// Mitsubishi GX Works2 project: PLC_Group12   PLC: FX3G

// global labels: Global1
VAR_GLOBAL
  switch7 AT X007 : BOOL;
  input_chocolate AT D1100 : REAL;
  reg_chocolate_container AT D1110 : REAL;
  reg_nuts_container AT D1112 : REAL;
  input_nuts AT D1102 : REAL;
  reg_pistachio_container AT D1114 : REAL;
  reg_kadaif_container AT D1116 : REAL;
  input_pistachio AT D1104 : REAL;
  input_kadaif AT D1106 : REAL;
  light7 AT Y007 : BOOL;
END_VAR
VAR_GLOBAL CONSTANT
  min_chocolate : REAL := 400.0;
  min_nuts : REAL := 100.0;
  min_pistachio : REAL := 120.0;
  min_kadaif : REAL := 60.0;
END_VAR
VAR_GLOBAL
  check_quantity AT M0 : BOOL;
  switch1 AT X001 : BOOL;
  melting_container AT D1120 : REAL;
  melting_process AT Y001 : BOOL;
  switch2 AT X002 : BOOL;
  switch3 AT X003 : BOOL;
  pouring AT TC1 : BOOL;
END_VAR
VAR_GLOBAL CONSTANT
  pouring_time : INT := 40;
END_VAR
VAR_GLOBAL
  pouring_light AT Y002 : BOOL;
  end_pouring AT TS1 : BOOL;
  switch4 AT X004 : BOOL;
  analog_input_1 AT D8280 : INT;
END_VAR
VAR_GLOBAL CONSTANT
  input_normalize : REAL := 400.0;
END_VAR
VAR_GLOBAL
  chocolate_choice AT D2000 : REAL;
END_VAR
VAR_GLOBAL CONSTANT
  min_choc_nuts : REAL;
  max_choc_nuts : REAL := 5.0;
END_VAR
VAR_GLOBAL
  choc_nuts_light AT M1 : BOOL;
END_VAR
VAR_GLOBAL CONSTANT
  max_choc_dubai : REAL := 10;
  min_choc_dubai : REAL := 5;
END_VAR
VAR_GLOBAL
  choc_dubai_light AT M2 : BOOL;
  pouring_container AT D1122 : REAL;
END_VAR
VAR_GLOBAL CONSTANT
  nuts_filler_for_nuts_choc : REAL := 100.0;
  pistachio_filler_for_nuts_choc : REAL := 100.0;
  nut_filler_for_dubai_choc : REAL := 20.0;
  pistachio_filler_for_dubai_choc : REAL := 120.0;
  kadaif_filler_for_dubai_choc : REAL := 60.0;
END_VAR
VAR_GLOBAL
  blinking3 AT M3 : BOOL;
  light3 AT Y003 : BOOL;
  blinking_switch_3 AT TS3 : BOOL;
  blinking_time_3 AT TC3 : BOOL;
  blinking_time_4 AT TC4 : BOOL;
END_VAR
VAR_GLOBAL CONSTANT
  blinking_time_limit_3 : INT := 10;
  blinking_time_limit_4 : INT := 10;
END_VAR
VAR_GLOBAL
  light4 AT Y004 : BOOL;
  blinking_switch_4 AT TS4 : BOOL;
  blinking_help_light_4 AT M4 : BOOL;
  blinking_help_light_5 AT TS5 : BOOL;
END_VAR
VAR_GLOBAL CONSTANT
  total_blinking_time : INT := 50;
END_VAR
VAR_GLOBAL
  blinking_time_5 AT TC5 : BOOL;
  switch6 AT X006 : BOOL;
  light6 AT Y006 : BOOL;
  cooling_switch AT TS6 : BOOL;
  cool_timer AT TC6 : BOOL;
END_VAR
VAR_GLOBAL CONSTANT
  cool_limit_time : WORD := 30;
END_VAR
VAR_GLOBAL
  switch0 AT X000 : BOOL;
  bars_counter AT CC0 : BOOL;
  bars_counter_switch AT CS0 : BOOL;
END_VAR
VAR_GLOBAL CONSTANT
  bars_limit : WORD := 4;
END_VAR
VAR_GLOBAL
  package_of_four_counter AT D1300 : REAL;
END_VAR
VAR_GLOBAL CONSTANT
  add_one_package : REAL := 1.0;
END_VAR
VAR_GLOBAL
  analog_output AT D8282 : INT;
END_VAR
VAR_GLOBAL CONSTANT
  zero_reset : REAL;
END_VAR
VAR_GLOBAL
  switch5 AT X005 : BOOL;
END_VAR
VAR_GLOBAL CONSTANT
  reset_chocolate_choice : REAL := 15.0;
END_VAR
VAR_GLOBAL
  process_1_done AT M11 : BOOL;
END_VAR
VAR_GLOBAL CONSTANT
  output_normalize : REAL := 40.0;
END_VAR
VAR_GLOBAL
  process_2_done AT M12 : BOOL;
  process_3_done AT M13 : BOOL;
  process_4_done AT M14 : BOOL;
  process_0_done AT M10 : BOOL;
  process_6_done AT M16 : BOOL;
  end_pouring_light AT M21 : BOOL;
  blinking_light_end AT M20 : BOOL;
  cool_light_end AT M22 : BOOL;
  choice_out_of_range AT M40 : BOOL;
  bars_packaging_light AT Y005 : BOOL;
END_VAR
VAR_GLOBAL CONSTANT
  devide_10_output : REAL := 10;
END_VAR

// task Task_01 (event TRUE, interval 0, priority 31): POU_01

PROGRAM POU_01
(* structured ladder/FBD written out as ST: instructions are called as NAME(EN, inputs, outputs); _pN, _eN, _tN stand for wires *)
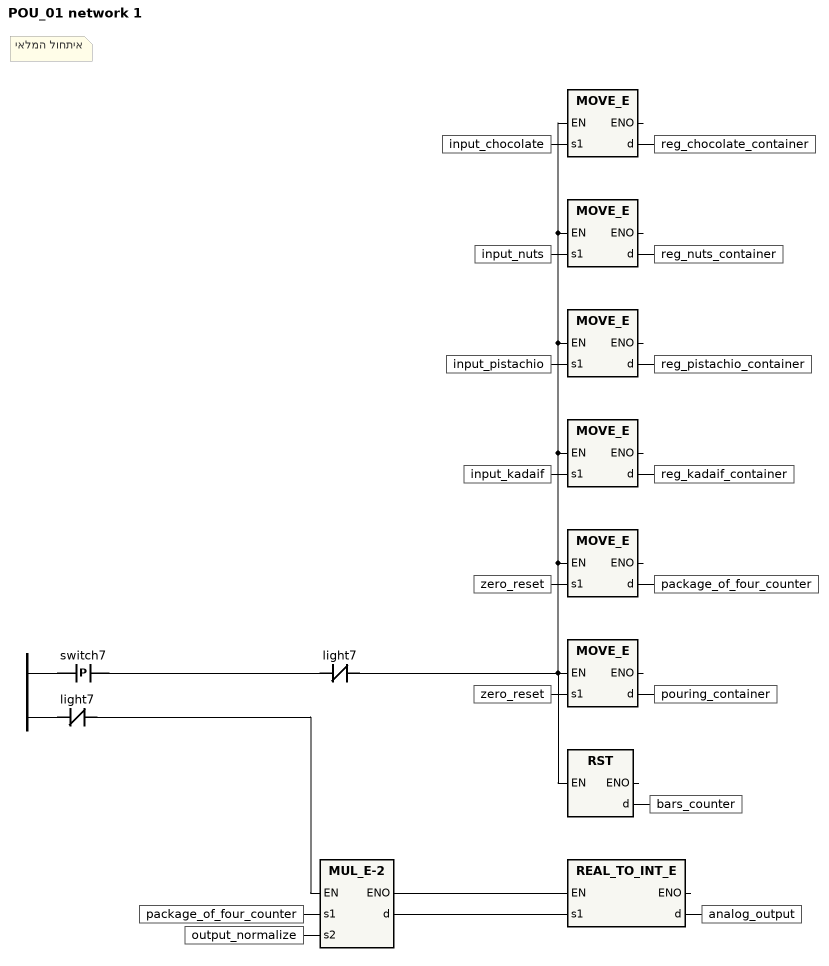
(* network 1 *)
(* איתחול המלאי *)
_p1 := LDP(TRUE, switch7) AND NOT light7;
MOVE_E(_p1, input_chocolate, reg_chocolate_container);
MOVE_E(_p1, input_nuts, reg_nuts_container);
MOVE_E(_p1, input_pistachio, reg_pistachio_container);
MOVE_E(_p1, input_kadaif, reg_kadaif_container);
MOVE_E(_p1, zero_reset, package_of_four_counter);
MOVE_E(_p1, zero_reset, pouring_container);
RST(_p1, bars_counter);
_e3 := MUL_E(NOT light7, package_of_four_counter, output_normalize, _t2);
REAL_TO_INT_E(_e3, _t2, analog_output);
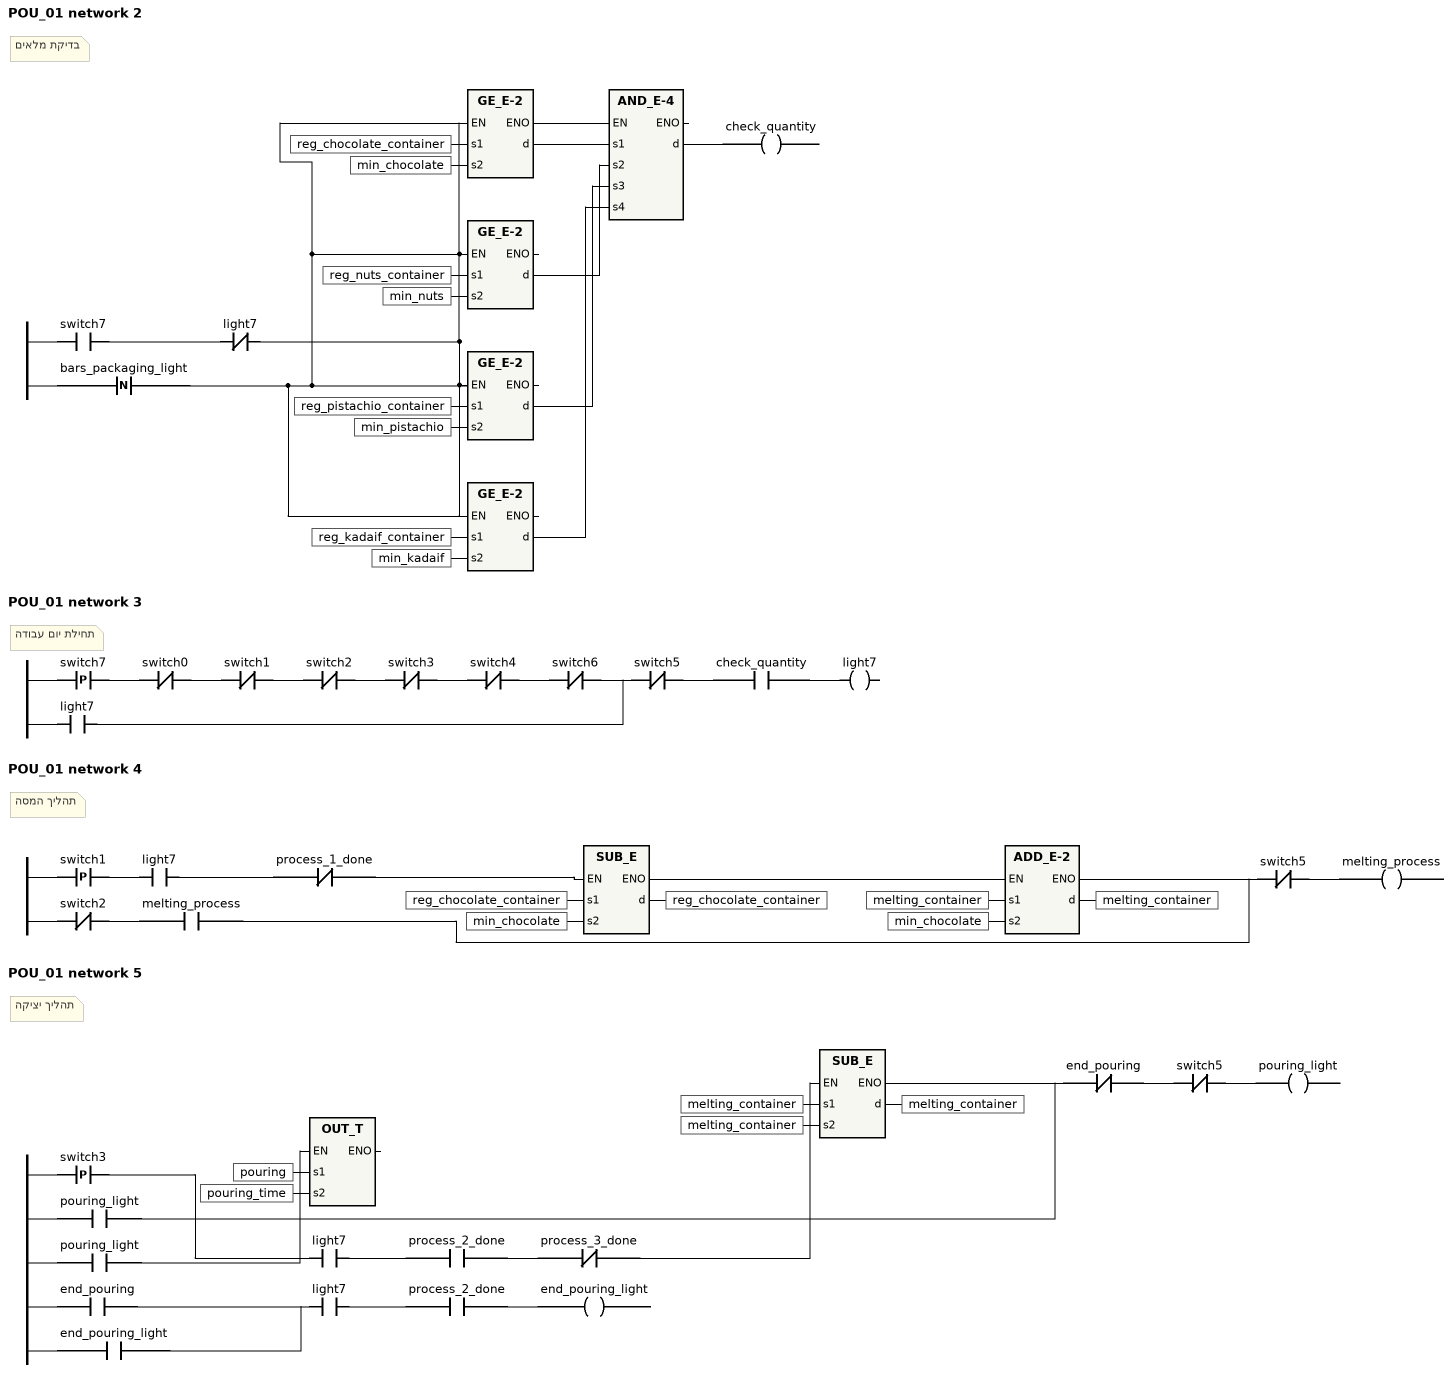
(* network 2 *)
(* בדיקת מלאים *)
_p1 := (switch7 AND NOT light7) OR LDF(TRUE, bars_packaging_light);
_e3 := GE_E(_p1, reg_chocolate_container, min_chocolate, _t2);
GE_E(_p1, reg_nuts_container, min_nuts, _t4);
GE_E(_p1, reg_pistachio_container, min_pistachio, _t5);
GE_E(_p1, reg_kadaif_container, min_kadaif, _t6);
AND_E(_e3, _t2, _t4, _t5, _t6, _t7);
check_quantity := _t7;
(* network 3 *)
(* תחילת יום עבודה *)
light7 := (((LDP(TRUE, switch7) AND NOT switch0 AND NOT switch1 AND NOT switch2 AND NOT switch3 AND NOT switch4 AND NOT switch6) OR light7) AND NOT switch5) AND check_quantity;
(* network 4 *)
(* תהליך המסה *)
_e1 := SUB_E(LDP(TRUE, switch1) AND light7 AND NOT process_1_done, reg_chocolate_container, min_chocolate, reg_chocolate_container);
_e2 := ADD_E(_e1, melting_container, min_chocolate, melting_container);
melting_process := (_e2 OR (NOT switch2 AND melting_process)) AND NOT switch5;
(* network 5 *)
(* תהליך יציקה *)
_e1 := SUB_E(LDP(TRUE, switch3) AND light7 AND process_2_done AND NOT process_3_done, melting_container, melting_container, melting_container);
pouring_light := ((_e1 OR pouring_light) AND NOT end_pouring) AND NOT switch5;
OUT_T(pouring_light, pouring, pouring_time);
end_pouring_light := ((end_pouring OR end_pouring_light) AND light7) AND process_2_done;
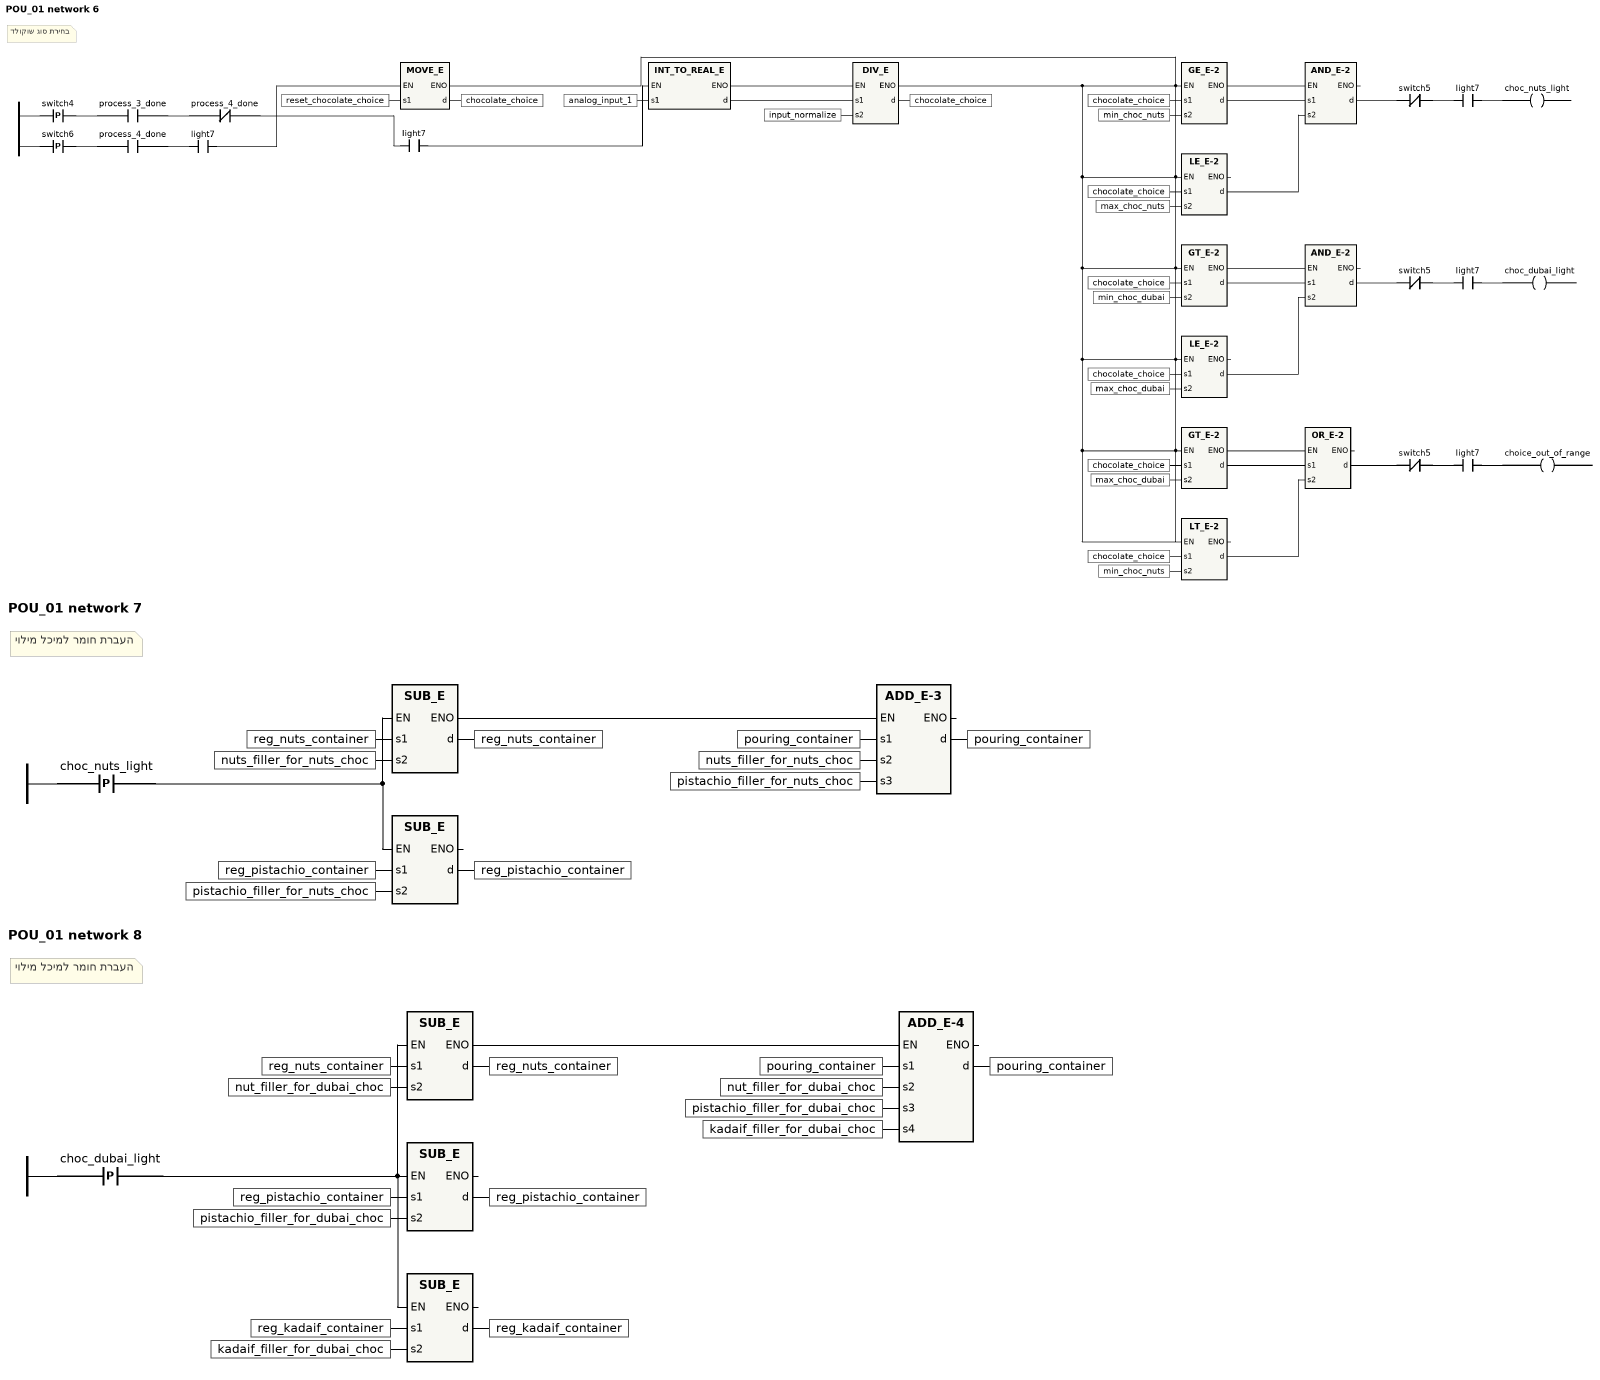
(* network 6 *)
(* בחירת סוג שוקולד *)
_e2 := INT_TO_REAL_E(LDP(TRUE, switch4) AND process_3_done AND NOT process_4_done AND light7, analog_input_1, _t1);
_e3 := DIV_E(_e2, _t1, input_normalize, chocolate_choice);
_e4 := MOVE_E(LDP(TRUE, switch6) AND process_4_done AND light7, reset_chocolate_choice, chocolate_choice);
_p5 := _e3 OR _e4;
_e7 := GE_E(_p5, chocolate_choice, min_choc_nuts, _t6);
LE_E(_p5, chocolate_choice, max_choc_nuts, _t8);
AND_E(_e7, _t6, _t8, _t9);
choc_nuts_light := _t9 AND NOT switch5 AND light7;
_e11 := GT_E(_p5, chocolate_choice, min_choc_dubai, _t10);
LE_E(_p5, chocolate_choice, max_choc_dubai, _t12);
AND_E(_e11, _t10, _t12, _t13);
choc_dubai_light := _t13 AND NOT switch5 AND light7;
_e15 := GT_E(_p5, chocolate_choice, max_choc_dubai, _t14);
LT_E(_p5, chocolate_choice, min_choc_nuts, _t16);
OR_E(_e15, _t14, _t16, _t17);
choice_out_of_range := _t17 AND NOT switch5 AND light7;
(* network 7 *)
(* העברת חומר למיכל מילוי *)
_p1 := LDP(TRUE, choc_nuts_light);
_e2 := SUB_E(_p1, reg_nuts_container, nuts_filler_for_nuts_choc, reg_nuts_container);
ADD_E(_e2, pouring_container, nuts_filler_for_nuts_choc, pistachio_filler_for_nuts_choc, pouring_container);
SUB_E(_p1, reg_pistachio_container, pistachio_filler_for_nuts_choc, reg_pistachio_container);
(* network 8 *)
(* העברת חומר למיכל מילוי *)
_p1 := LDP(TRUE, choc_dubai_light);
_e2 := SUB_E(_p1, reg_nuts_container, nut_filler_for_dubai_choc, reg_nuts_container);
ADD_E(_e2, pouring_container, nut_filler_for_dubai_choc, pistachio_filler_for_dubai_choc, kadaif_filler_for_dubai_choc, pouring_container);
SUB_E(_p1, reg_pistachio_container, pistachio_filler_for_dubai_choc, reg_pistachio_container);
SUB_E(_p1, reg_kadaif_container, kadaif_filler_for_dubai_choc, reg_kadaif_container);
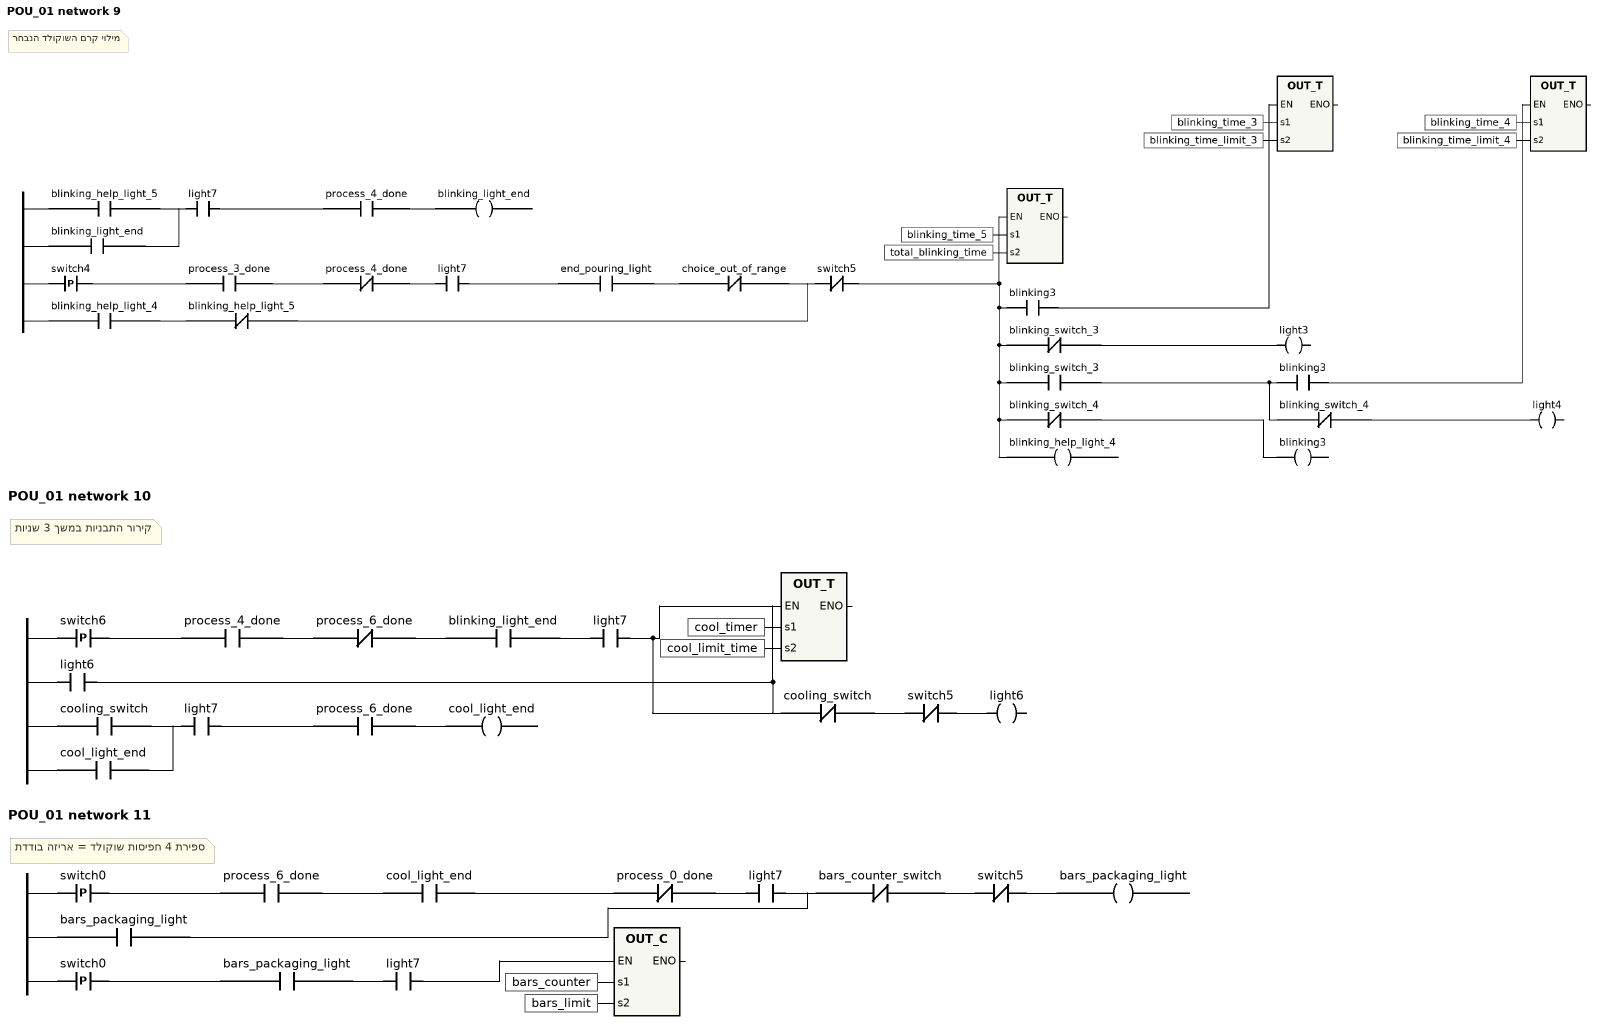
(* network 9 *)
(* מילוי קרם השוקולד הנבחר *)
blinking_light_end := ((blinking_help_light_5 OR blinking_light_end) AND light7) AND process_4_done;
_p1 := ((LDP(TRUE, switch4) AND process_3_done AND NOT process_4_done AND light7 AND end_pouring_light AND NOT choice_out_of_range) OR (blinking_help_light_4 AND NOT blinking_help_light_5)) AND NOT switch5;
OUT_T(_p1 AND blinking3, blinking_time_3, blinking_time_limit_3);
light3 := _p1 AND NOT blinking_switch_3;
_p2 := _p1 AND blinking_switch_3;
OUT_T(_p2 AND blinking3, blinking_time_4, blinking_time_limit_4);
light4 := _p2 AND NOT blinking_switch_4;
OUT_T(_p1, blinking_time_5, total_blinking_time);
blinking3 := _p1 AND NOT blinking_switch_4;
blinking_help_light_4 := _p1;
(* network 10 *)
(* קירור התבניות במשך 3 שניות *)
_p1 := (LDP(TRUE, switch6) AND process_4_done AND NOT process_6_done AND blinking_light_end AND light7) OR light6;
light6 := _p1 AND NOT cooling_switch AND NOT switch5;
OUT_T(_p1, cool_timer, cool_limit_time);
cool_light_end := ((cooling_switch OR cool_light_end) AND light7) AND process_6_done;
(* network 11 *)
(* ספירת 4 חפיסות שוקולד = אריזה בודדת *)
bars_packaging_light := (((LDP(TRUE, switch0) AND process_6_done AND cool_light_end AND NOT process_0_done AND light7) OR bars_packaging_light) AND NOT bars_counter_switch) AND NOT switch5;
OUT_C(LDP(TRUE, switch0) AND bars_packaging_light AND light7, bars_counter, bars_limit);
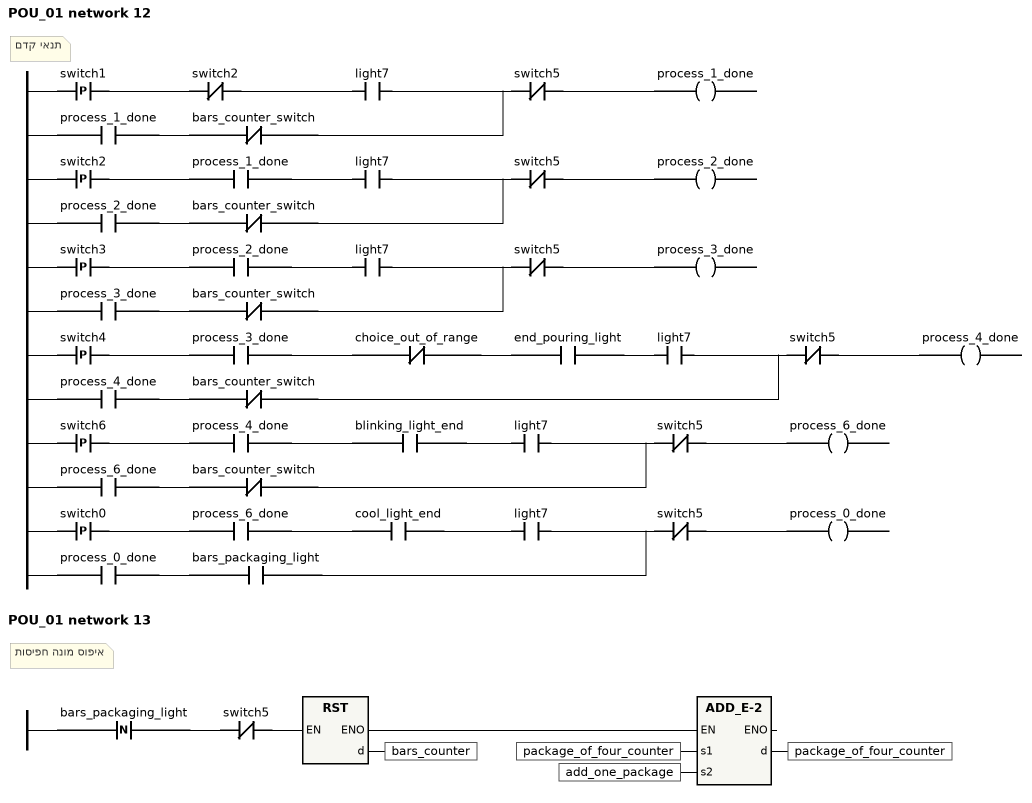
(* network 12 *)
(* תנאי קדם *)
process_1_done := ((LDP(TRUE, switch1) AND NOT switch2 AND light7) OR (process_1_done AND NOT bars_counter_switch)) AND NOT switch5;
process_2_done := ((LDP(TRUE, switch2) AND process_1_done AND light7) OR (process_2_done AND NOT bars_counter_switch)) AND NOT switch5;
process_3_done := ((LDP(TRUE, switch3) AND process_2_done AND light7) OR (process_3_done AND NOT bars_counter_switch)) AND NOT switch5;
process_4_done := ((LDP(TRUE, switch4) AND process_3_done AND NOT choice_out_of_range AND end_pouring_light AND light7) OR (process_4_done AND NOT bars_counter_switch)) AND NOT switch5;
process_6_done := ((LDP(TRUE, switch6) AND process_4_done AND blinking_light_end AND light7) OR (process_6_done AND NOT bars_counter_switch)) AND NOT switch5;
process_0_done := ((LDP(TRUE, switch0) AND process_6_done AND cool_light_end AND light7) OR (process_0_done AND bars_packaging_light)) AND NOT switch5;
(* network 13 *)
(* איפוס מונה חפיסות *)
_e1 := RST(LDF(TRUE, bars_packaging_light) AND NOT switch5, bars_counter);
ADD_E(_e1, package_of_four_counter, add_one_package, package_of_four_counter);
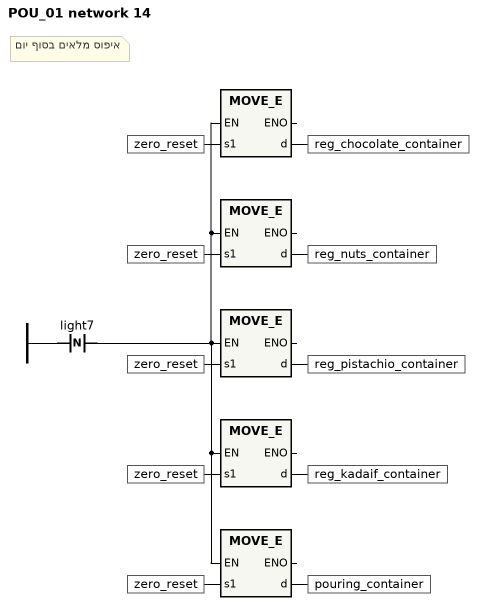
(* network 14 *)
(* איפוס מלאים בסוף יום *)
_p1 := LDF(TRUE, light7);
MOVE_E(_p1, zero_reset, reg_chocolate_container);
MOVE_E(_p1, zero_reset, reg_nuts_container);
MOVE_E(_p1, zero_reset, reg_pistachio_container);
MOVE_E(_p1, zero_reset, reg_kadaif_container);
MOVE_E(_p1, zero_reset, pouring_container);
END_PROGRAM
